// TIA Portal V20 export
// export: Created 2025-12-01T14:56:14.3321754Z, ExportSetting None, DisplayName Totally Integrated Automation Portal, DisplayVersion V20 Update 3, DisplayName TIA Portal Openness, DisplayVersion V20 Update 3, DisplayName TIA Portal Version Control Interface, DisplayVersion V20 Update 3, DisplayName STEP 7 Professional, DisplayVersion V20 Update 3, DisplayName STEP 7 Safety, DisplayVersion V20 Update 2, DisplayName WinCC Basic/Comfort/Advanced, DisplayVersion V20 Update 3, DisplayName WinCC Professional, DisplayVersion V20 Update 3, DisplayName WinCC Unified, DisplayVersion V20 Update 3
TYPE "UDT_DefinicionMesa"
   STRUCT
      Mesa_S01 : UInt;   // Mesa con salida en S01
      Mesa_S02 : UInt;   // Mesa con salida en S02
      Mesa_S03 : UInt;   // Mesa con salida en S03
      Mesa_S04 : UInt;   // Mesa con salida en S04
      AtributosGalibo_Guardar : Struct   // Galibo a Guardar en la Mesa (Programa)
         Altura : Bool;   // Codigo de Altura
         Anchura : Bool;   // Codigo de Anchura
         Profundidad : Bool;   // Codigo de Profundidad
         Taco : Bool;   // Codigo de Taco
         Hueco : Bool;   // Codigo de Hueco
         HuecoRemontado : Bool;   // Codigo de Hueco para Paleta Remontada
         Color : Bool;   // Codigo de Color
         Patin : Bool;   // Codigo de Patin
         Tipo : Bool;   // Codigo de Tipo de Carga
         Remontado : Bool;   // Codigo de Paleta Remontada
         Cota_Altura : Bool;   // Cota de Altura
         Cota_Anchura : Bool;   // Cota de Anhura
         Cota_Profundidad : Bool;   // Cota de Profundidad
         Peso : Bool;   // Peso
         EtiquetaRouter : Bool;   // Etiqueta del Router
         EtiquetaString : Bool;   // Etiqueta en formato String
      END_STRUCT;
      AtributosGalibo_DeEvento : Struct   // Galibo a Enviar en la Mesa (Evento)
         Altura : Bool;   // Codigo de Altura
         Anchura : Bool;   // Codigo de Anchura
         Profundidad : Bool;   // Codigo de Profundidad
         Taco : Bool;   // Codigo de Taco
         Hueco : Bool;   // Codigo de Hueco
         HuecoRemontado : Bool;   // Codigo de Hueco para Paleta Remontada
         Color : Bool;   // Codigo de Color
         Patin : Bool;   // Codigo de Patin
         Tipo : Bool;   // Codigo de Tipo de Carga
         Remontado : Bool;   // Codigo de Paleta Remontada
         Cota_Altura : Bool;   // Cota de Altura
         Cota_Anchura : Bool;   // Cota de Anhura
         Cota_Profundidad : Bool;   // Cota de Profundidad
         Peso : Bool;   // Peso
         EtiquetaRouter : Bool;   // Etiqueta del Router
         EtiquetaString : Bool;   // Etiqueta en formato String
      END_STRUCT;
      ConfigMesa : Struct   // Definicion de la Mesa (Sistema)
         TipoMaquina : UInt := 70;   // Tipo de Maquina existente en la Mesa
         MesaPaso : Bool;   // Es una mesa de Paso
         MesaCruce : Bool;   // Es una mesa de Cruce
         MesaMultiplesDestinos : Bool;   // Es una mesa de Multiples Destinos (1º MESA de la Ruta)
         MesaTL : Bool;   // Es mesa de TL
         MaquinaEnMesa : Bool;   // Existe Maquina en la Mesa
         MesaDeJDT02 : Bool;   // Mesa Pertenciente a la conexion del JDT02
         MultipleCapacidad : Bool;   // Capacidad de la Mesa de mas de Una UT en la Mesa
         PeticionDeDatos : Bool;   // Pedir Datos de la UT Adicionales al JDT
         SinPresenciaEnReset : Bool;   // No se envia presencia en el Reset (Parcial)
         MeterAlPrincipio : Bool;   // Sirve para el cambio de Mesa (Insertar al Final o Al Principio)
         SinErrorDeDatosVacia : Bool;   // Sin el Error de Datos de la Mesa cuando esta Vacia
         SinErrorDeDatosCargada : Bool;   // Sin el Error de Datos de la Mesa cuando esta Cargada
         NoInformar : Bool;   // No Informar al JdT
         EspecialOrdenes : Bool;   // Es una mesa que tiene su propio generador de ordenes
         RutaSalidaTodas : Bool;   // Tienen todas las UT's Destino
         AusenciaMultiple : Bool;   // Es una mesa que la ausencia es para todas las UT's de la Mesa
         AusenciaBorrarUT : Bool;   // Con la Ausencia se debe BORRAR la UT y no emviar el RETI
         GrupoDeSalida : Bool;   // Grupo de Cargas de Salida
         MultiplesCargasDeSalida : Bool;   // Multiples Cargas de Salida
         GrupoDeEntrada : Bool;   // Grupo de Cargas de Entrada
         MultiplesCargasDeEntrada : Bool;   // Multiples Cargas de Entrada
         Espera_S01 : Bool;   // Espera que la Mesa Siguiente no tenga UT's, Salida S01
         Espera_S02 : Bool;   // Espera que la Mesa Siguiente no tenga UT's, Salida S02
         Espera_S03 : Bool;   // Espera que la Mesa Siguiente no tenga UT's, Salida S03
         Espera_S04 : Bool;   // Espera que la Mesa Siguiente no tenga UT's, Salida S04
      END_STRUCT;
      ConfigFB { S7_SetPoint := 'True'} : "UDT_ConfigFB";   // Definicion de la Mesa para las FBs
   END_STRUCT;
END_TYPE
